TEXTLIST M3ConfigTabsTextList
  0 = 'General'
  1 = 'Known positions'
  2 = 'Rotation - general'
  3 = 'Rotation - positioning drive'
  4 = 'Rotation - anti-backlash drive'
  5 = 'Translation - general'
  6 = 'Translation - drive'
   = ''
END_TEXTLIST

(* stored: Version 1.1.0.1, ProductVersion 3.1.4018.5
   TextList M3ConfigTabsTextList: Id {be4501c5-f0b8-40d8-8aaf-c9c297a14696} *)
